Fanuc KAREL source: compact_preamble.KL

PROGRAM KX00028
%TIMESLICE=8
%NOLOCKGROUP
VAR
I:INTEGER;J:INTEGER;B:BOOLEAN
F : FILE
S : STRING[80]
P : XYZWPR
BEGIN
I=1
END KX00028
